Staubli VAL3: writeSocket.pgx

program writeSocket(num x_nCamID (dimensions=1), string x_sMsg (dimensions=1))
  local num i
begin
  //-----------------------------------------------------------------------
  //Header begin
  //Description of program
  //  Write string to socket character by character.
  //
  //Input parameters
  //  num x_nCamID :
  //    role : camera's ID
  //  string x_sMsg :
  //    role : native command
  //
  //Examples
  //  call sendCommand(nCamID,sCmd)
  //
  //History
  //  Creation : 19-05-08 - f.Rob
  //Header end
  //-----------------------------------------------------------------------

  for i=0 to (len(x_sMsg)-1)
    sioSet(cCamera[x_nCamID].sSocket,asc(x_sMsg,i))
  endFor
  sioSet(cCamera[x_nCamID].sSocket,13)
  sioSet(cCamera[x_nCamID].sSocket,10)
  if bDebugSocket
    ? "W Status code: "+x_sMsg
  endIf
end
